INTERFACE I_PackML_SuspendedCommands

METHOD PUBLIC Abort
VAR_INPUT
END_VAR
END_METHOD

METHOD PUBLIC Stop
VAR_INPUT
END_VAR
END_METHOD

METHOD PUBLIC Unsuspend
VAR_INPUT
END_VAR
END_METHOD

END_INTERFACE

(* stored: Version 1.1.0.1, ProductVersion 3.1.4024.12
   Itf I_PackML_SuspendedCommands: Id {f31c0d5b-acac-0491-1bc4-9e5110404f07}
   Method Abort: Id {c2b501bc-2d8c-086e-3fd9-ac173dc4eff0}
   Method Stop: Id {297816d5-de90-0d80-371d-a6f5129a6bb2}
   Method Unsuspend: Id {199c3e50-b73d-0b1c-0fc2-c7e590019e1b} *)
